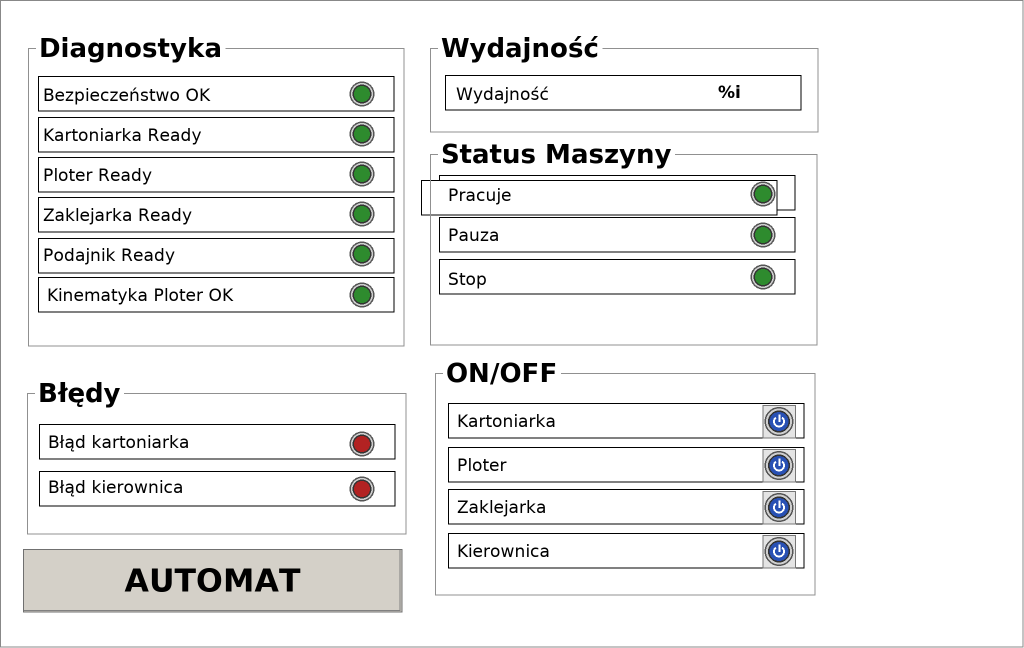
VISUALIZATION Glowna  // 1024x648
    Rectangle (439,175 356x35)
    GroupBox (28,40 376x306), "Diagnostyka"
        Rectangle (10,198 356x35)
        Rectangle (10,157 356x35)
        Rectangle (10,117 356x35)
        Rectangle (10,77 356x35)
        Rectangle (10,36 356x35)
        Label (12,40 209x30), "Bezpieczeństwo OK"
        Label (12,80 209x30), "Kartoniarka Ready"
        Label (12,160 209x30), "Zaklejarka Ready"
        Label (12,200 209x30), "Podajnik Ready"
        Lamp1 (320,40 28x28), variable: GVL_SafetyFrom_RT2.bSAFETY_PermissionSS1 and GVL_SafetyFrom_RT2.bSAFETY_PermissionSS2, style: Lamp-Lamp1-Green
        Lamp1 (320,80 28x28), style: Lamp-Lamp1-Green
        Lamp1 (320,120 28x28), style: Lamp-Lamp1-Green
        Lamp1 (320,200 28x28), style: Lamp-Lamp1-Green
        Lamp1 (320,160 28x28), style: Lamp-Lamp1-Green
        Rectangle (10,237 356x35)
        Label (16,240 209x30), "Kinematyka Ploter OK"
        Lamp1 (320,241 28x28), style: Lamp-Lamp1-Green
        Label (12,120 209x30), "Ploter Ready"
        Rectangle (393,140 356x35)
    GroupBox (430,40 388x92), "Wydajność"
        Rectangle (15,35 356x35)
        Label (23,39 209x30), "Wydajność"
        Label (209,101 100x25)
        Textfield (239,37 121x30), "%i", text variable: GVL_HMI.iWydajnosc
    GroupBox (435,365 380x230), "ON/OFF"
        Rectangle (13,38 356x35)
        Label (19,41 209x30), "Kartoniarka"
        Rectangle (13,82 356x35)
        Label (19,85 209x30), "Ploter"
        Rectangle (13,168 356x35)
        Label (19,171 209x30), "Kierownica"
        Rectangle (13,124 356x35)
        Label (19,127 209x30), "Zaklejarka"
        PowerSwitch (325,40 38x33), variable: GVL_HMI.bEnableKartoniarka, behaviour: TOGGLE, style: Switch-PowerSwitch-Blue
        PowerSwitch (325,84 38x33), variable: GVL_HMI.bEnablePloter, behaviour: TOGGLE, style: Switch-PowerSwitch-Blue
        PowerSwitch (325,126 38x33), variable: GVL_HMI.bEnableZaklejarka, behaviour: TOGGLE, style: Switch-PowerSwitch-Blue
        PowerSwitch (325,170 38x33), variable: GVL_HMI.bEnableKierownica, behaviour: TOGGLE, style: Switch-PowerSwitch-Blue
    GroupBox (430,146 387x199), "Status Maszyny"
        Label (211,97 100x25)
    Label (445,180 209x30), "Pracuje"
    Lamp1 (749,180 28x28), style: Lamp-Lamp1-Green
    Rectangle (439,217 356x35)
    Label (445,220 209x30), "Pauza"
    Lamp1 (749,221 28x28), style: Lamp-Lamp1-Green
    Rectangle (439,259 356x35)
    Label (445,264 209x30), "Stop"
    Lamp1 (749,263 28x28), style: Lamp-Lamp1-Green
    GroupBox (27,385 379x149), "Błędy"
        Textfield (240,41 121x30), text variable: GVL_HMI.INT_idError
        Rectangle (12,39 356x35)
        Label (18,42 209x30), "Błąd kartoniarka"
        Lamp1 (321,45 28x28), variable: GVL_GLOBAL.Error_ind_kart, style: Lamp-Lamp1-Red
        Rectangle (12,86 356x35)
        Lamp1 (321,90 28x28), variable: GVL_GLOBAL.Error_pakowania, style: Lamp-Lamp1-Red
        Label (18,87 209x30), "Błąd kierownica"
    Button (23,549 379x63), "AUTOMAT"
        toggle GVL_HMI.bAutoWybor
END_VISUALIZATION

(* stored: Version 1.1.0.1, ProductVersion 3.1.4022.12
   Visu Glowna: Id {e17900c9-3696-44f3-b4c8-001e233847e1} *)
